// TIA Portal V16 export
// export: Created 2025-12-18T09:29:18.7941412Z, ExportSetting WithDefaults, DisplayName Totally Integrated Automation Portal, DisplayVersion V16, DisplayName TIA Portal Version Control Interface, DisplayVersion V16, DisplayName TIA Portal Openness, DisplayVersion V16, DisplayName STEP 7 Professional, DisplayVersion V16, DisplayName STEP 7 Safety, DisplayVersion V16, DisplayName WinCC Advanced, DisplayVersion V16
VAR_GLOBAL   // PLC tag table "Outputs"
   qIO_xSupplyConveyor1 AT %Q0.0 : Bool;
   qIO_xSupplyConveyor2 AT %Q0.1 : Bool;
   qIO_xS1Conveyor1 AT %Q0.2 : Bool;
   qIO_xS1Conveyor2 AT %Q0.3 : Bool;
   qIO_xS1Conveyor3 AT %Q0.4 : Bool;
   qIO_xS1PositionerClamp AT %Q0.5 : Bool;
   qIO_xS1PositionerRaise AT %Q0.6 : Bool;
   qIO_xS2Conveyor1 AT %Q0.7 : Bool;
   qIO_xS2Conveyor2 AT %Q1.0 : Bool;
   qIO_xS2Conveyor3 AT %Q1.1 : Bool;
   qIO_xS2PositionerClamp AT %Q1.2 : Bool;
   qIO_xS2PositionerRaise AT %Q1.3 : Bool;
   qIO_xS3Conveyor1 AT %Q1.4 : Bool;
   qIO_xS3Conveyor2 AT %Q1.5 : Bool;
   qIO_xS3Conveyor3 AT %Q1.6 : Bool;
   qIO_xS3PositionerClamp AT %Q1.7 : Bool;
   qIO_xS3PositionerRaise AT %Q2.0 : Bool;
   qIO_xS1ProcessLight AT %Q2.1 : Bool;
   qIO_iS1ProcessTimeLeft AT %QD10 : DInt;
   qIO_xS2ProcessLight AT %Q2.2 : Bool;
   qIO_iS2ProcessTimeLeft AT %QD14 : DInt;
   qIO_xS3ProcessLight AT %Q2.3 : Bool;
   qIO_iS3ProcessTimeLeft AT %QD18 : DInt;
   qIO_xSupplyGetMaterial AT %Q2.4 : Bool;
END_VAR
